// TIA Portal V17 export
// export: Created 2025-04-11T04:54:23.8282956Z, ExportSetting WithDefaults, DisplayName Totally Integrated Automation Portal, DisplayVersion V17, DisplayName TIA Portal Openness, DisplayVersion V17, DisplayName TIA Portal Version Control Interface, DisplayVersion V17, DisplayName SINAMICS Startdrive Advanced, DisplayVersion V17, DisplayName SINAMICS Startdrive G130, G150, S120, S150, SINAMICS MV, S210, DisplayVersion V17, DisplayName SINAMICS Startdrive G110M, G120, G120C, G120D, G120P, G115D, DisplayVersion V17, DisplayName STEP 7 Professional, DisplayVersion V17, DisplayName STEP 7 Safety, DisplayVersion V17, DisplayName WinCC Advanced, DisplayVersion V17
TYPE "UDT_Device_Map"
// stored: IsFailsafeCompliant false
   STRUCT
      IN_xStartFeedback : Bool;   // 设备启动反馈
      IN_xAlarmFeedback : Bool;   // 设备报警反馈
      OUT_xActualOut : Bool;   // 设备控制
      OUT_xStartDevice : Bool;   // 启动对方设备信号（上升沿有效，1秒后自动复位）
      OUT_xStopDevice : Bool;   // 停止对方设备信号（下降沿有效，1秒后自动复位）
   END_STRUCT;
END_TYPE
